Omron CX-Programmer project NewProject (CX-Programmer 9.73)

# PLC NewPLC1: CP1E N20

## Global symbols (name address type ; comment)
0.01 BOOL  ; PB START
100.00 BOOL  ; OUTPUT
T001 BOOL  ; PERMASA

## Program NewProgram1 (cyclic task 0)

### Section Section1

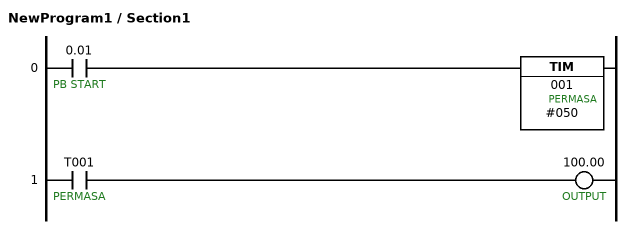
; rung 0
LD 0.01  ; PB START
TIM 001 #050  ; PERMASA
; rung 1
LD T001  ; PERMASA
OUT 100.00  ; OUTPUT

### Section END
; rung 0
END(001)